// TIA Portal V17 export
// export: Created 2025-06-26T06:49:12.8721557Z, ExportSetting WithDefaults, DisplayName Totally Integrated Automation Portal, DisplayVersion V17 Update 8, DisplayName TIA Portal Openness, DisplayVersion V17 Update 8, DisplayName TIA Portal Version Control Interface, DisplayVersion V17, DisplayName STEP 7 Professional, DisplayVersion V17 Update 8, DisplayName STEP 7 Safety, DisplayVersion V17 Update 6, DisplayName WinCC Advanced, DisplayVersion V17 Update 8
FUNCTION_BLOCK "OilSeparator"   // FB15, FBD
TITLE = Oil Separator
{ S7_Optimized_Access := 'TRUE' }
VERSION : 0.1
// stored: AutoNumber true, IsIECCheckEnabled false, IsRetainMemResEnabled false, MemoryReserve 100, SetENOAutomatically false, UDAEnableTagReadback false
   VAR_INPUT
      bEnable { ExternalAccessible := 'False'; ExternalVisible := 'False'; ExternalWritable := 'False'} : Bool;
      bReset { ExternalAccessible := 'False'; ExternalVisible := 'False'; ExternalWritable := 'False'} : Bool;   // 1 = reset manual modes
   END_VAR
   VAR
      Regulator { ExternalAccessible := 'False'; ExternalVisible := 'False'; ExternalWritable := 'False'} : "fbOnOffRegulator";
      Alarm { ExternalAccessible := 'False'; ExternalVisible := 'False'; ExternalWritable := 'False'; S7_SetPoint := 'True'} : "fbDigitalAlarm";
      Stage1 { S7_SetPoint := 'True'} : "fbOnOffRegulator2";
      Stage2 { S7_SetPoint := 'True'} : "fbOnOffRegulator2";
   END_VAR
   VAR_TEMP
      Enabled : Bool;
   END_VAR
BEGIN

REGION Network 1: Stage 1 level control
   // Run only when the pressure in oil separator Stage 1 is greater than the oil sump, so oil will move from oil separator to sump
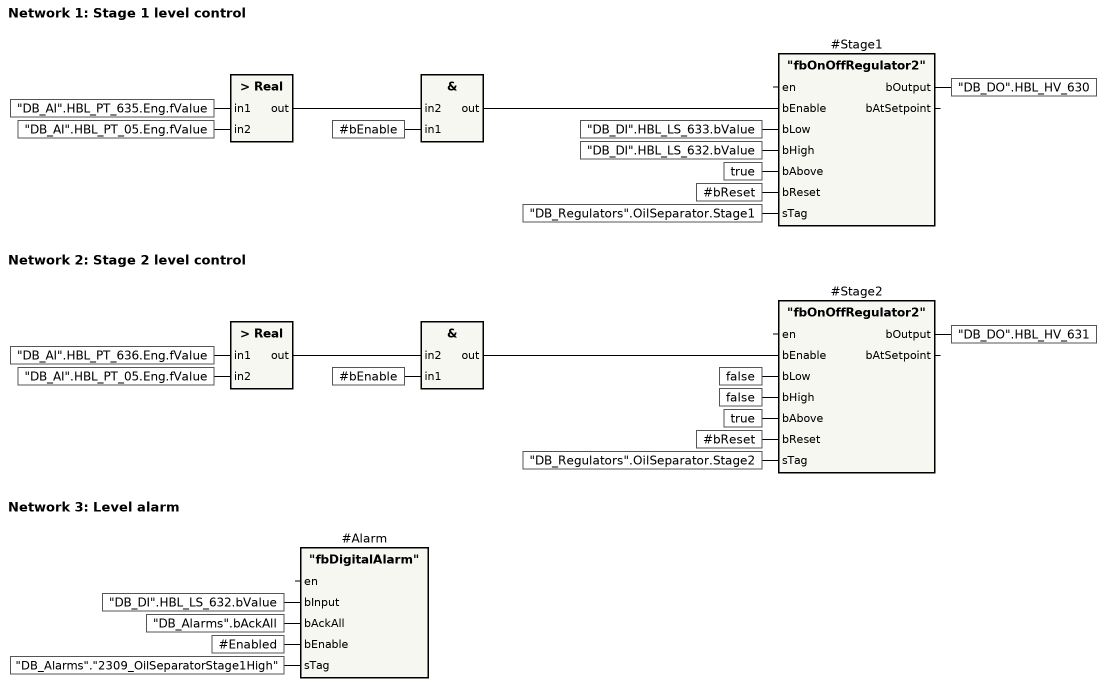
   #Stage1(bEnable := ("DB_AI".HBL_PT_635.Eng.fValue > "DB_AI".HBL_PT_05.Eng.fValue) AND #bEnable,   // "fbOnOffRegulator2"
           bLow := "DB_DI".HBL_LS_633.bValue,
           bHigh := "DB_DI".HBL_LS_632.bValue,
           bAbove := true,
           bReset := #bReset,
           sTag := "DB_Regulators".OilSeparator.Stage1,
           bOutput => "DB_DO".HBL_HV_630);
END_REGION

REGION Network 2: Stage 2 level control
   // Run only when the pressure in oil separator Stage 2 is greater than the oil sump, so oil will move from oil separator to sump
   // 10.02.2025 TSS: Currently no level switches in the P&ID, not sure of the control strategy
   #Stage2(bEnable := ("DB_AI".HBL_PT_636.Eng.fValue > "DB_AI".HBL_PT_05.Eng.fValue) AND #bEnable,   // "fbOnOffRegulator2"
           bLow := false,
           bHigh := false,
           bAbove := true,
           bReset := #bReset,
           sTag := "DB_Regulators".OilSeparator.Stage2,
           bOutput => "DB_DO".HBL_HV_631);
END_REGION

REGION Network 3: Level alarm
   // High level for a long time is probably worth knowing about
   #Alarm(bInput := "DB_DI".HBL_LS_632.bValue,   // "fbDigitalAlarm"
          bAckAll := "DB_Alarms".bAckAll,
          bEnable := #Enabled,
          sTag := "DB_Alarms"."2309_OilSeparatorStage1High");
END_REGION
END_FUNCTION_BLOCK
